# EPICS substitutions: mc06/tpmacApp/Db/autohome.substitutions
file "$(EPICS_BASE)/db/autohome.db"
{

pattern
{SYS           , DEV              , PLC , PORT  }
{"XF:23ID1-BI" , "{Diag:4-Ax:Y}"  , 8   , P0    }
{"XF:23ID1-OP" , "{Sh:Fast-Ax:Y}" , 9   , P0    }
{"XF:23ID1-OP" , "{Sh:Fast-Ax:X}" , 10  , P0    }
{"XF:23ID1-BI" , "{Diag:6-Ax:Y}"  , 11  , P0    }
}
